// LS Electric XG5000 project: FactoryIO_Automated Warehouse
// PLC LSPLC

PROGRAM NewProgram (task: 스캔 프로그램)

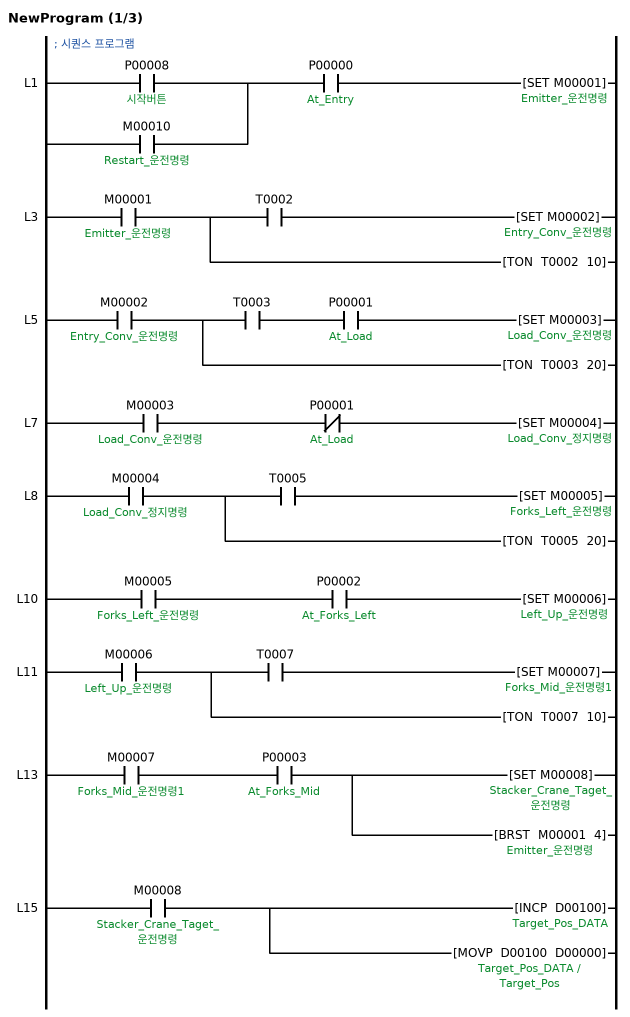
// 시퀀스 프로그램
; L1
LOAD      P00008	// 시작버튼
OR        M00010	// Restart_운전명령
AND       P00000	// At_Entry
SET       M00001	// Emitter_운전명령
; L3
LOAD      M00001	// Emitter_운전명령
MPUSH
AND       T0002
SET       M00002	// Entry_Conv_운전명령
MPOP
TON       T0002 10
; L5
LOAD      M00002	// Entry_Conv_운전명령
MPUSH
AND       T0003
AND       P00001	// At_Load
SET       M00003	// Load_Conv_운전명령
MPOP
TON       T0003 20
; L7
LOAD      M00003	// Load_Conv_운전명령
AND NOT   P00001	// At_Load
SET       M00004	// Load_Conv_정지명령
; L8
LOAD      M00004	// Load_Conv_정지명령
MPUSH
AND       T0005
SET       M00005	// Forks_Left_운전명령
MPOP
TON       T0005 20
; L10
LOAD      M00005	// Forks_Left_운전명령
AND       P00002	// At_Forks_Left
SET       M00006	// Left_Up_운전명령
; L11
LOAD      M00006	// Left_Up_운전명령
MPUSH
AND       T0007
SET       M00007	// Forks_Mid_운전명령1
MPOP
TON       T0007 10
; L13
LOAD      M00007	// Forks_Mid_운전명령1
AND       P00003	// At_Forks_Mid
SET       M00008	// Stacker_Crane_Taget_운전명령
BRST      M00001 4	// Emitter_운전명령
; L15
LOAD      M00008	// Stacker_Crane_Taget_운전명령
INCP      D00100	// Target_Pos_DATA
MOVP      D00100 D00000	// Target_Pos_DATA / Target_Pos

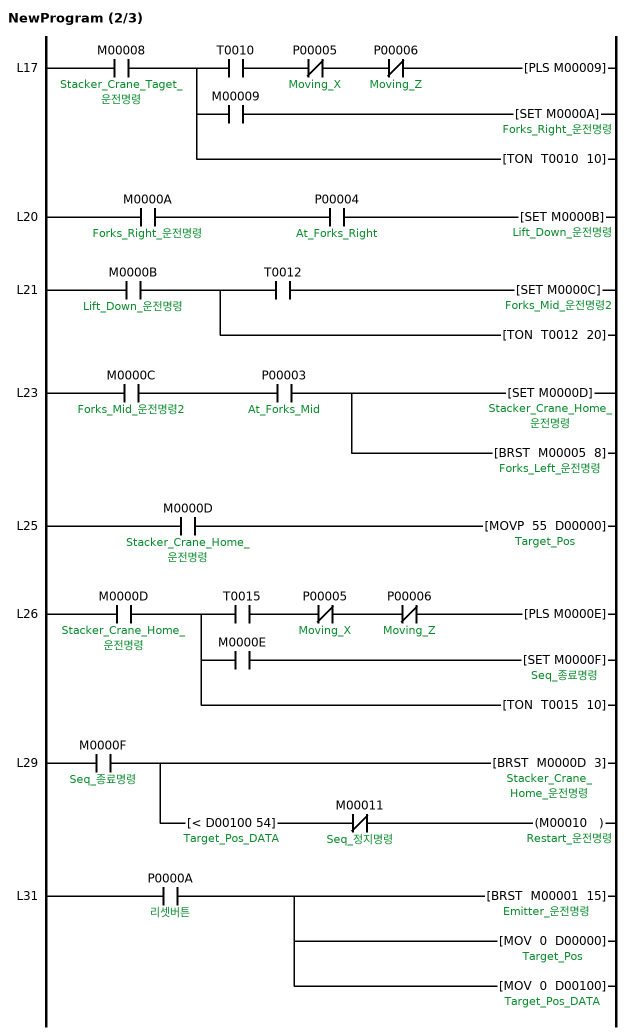
; L17
LOAD      M00008	// Stacker_Crane_Taget_운전명령
MPUSH
AND       T0010
AND NOT   P00005	// Moving_X
AND NOT   P00006	// Moving_Z
OUTP      M00009
MLOAD
AND       M00009
SET       M0000A	// Forks_Right_운전명령
MPOP
TON       T0010 10
; L20
LOAD      M0000A	// Forks_Right_운전명령
AND       P00004	// At_Forks_Right
SET       M0000B	// Lift_Down_운전명령
; L21
LOAD      M0000B	// Lift_Down_운전명령
MPUSH
AND       T0012
SET       M0000C	// Forks_Mid_운전명령2
MPOP
TON       T0012 20
; L23
LOAD      M0000C	// Forks_Mid_운전명령2
AND       P00003	// At_Forks_Mid
SET       M0000D	// Stacker_Crane_Home_운전명령
BRST      M00005 8	// Forks_Left_운전명령
; L25
LOAD      M0000D	// Stacker_Crane_Home_운전명령
MOVP      55 D00000	// Target_Pos
; L26
LOAD      M0000D	// Stacker_Crane_Home_운전명령
MPUSH
AND       T0015
AND NOT   P00005	// Moving_X
AND NOT   P00006	// Moving_Z
OUTP      M0000E
MLOAD
AND       M0000E
SET       M0000F	// Seq_종료명령
MPOP
TON       T0015 10
; L29
LOAD      M0000F	// Seq_종료명령
BRST      M0000D 3	// Stacker_Crane_Home_운전명령
AND<      D00100 54	// Target_Pos_DATA
AND NOT   M00011	// Seq_정지명령
OUT       M00010	// Restart_운전명령
; L31
LOAD      P0000A	// 리셋버튼
BRST      M00001 15	// Emitter_운전명령
MOV       0 D00000	// Target_Pos
MOV       0 D00100	// Target_Pos_DATA

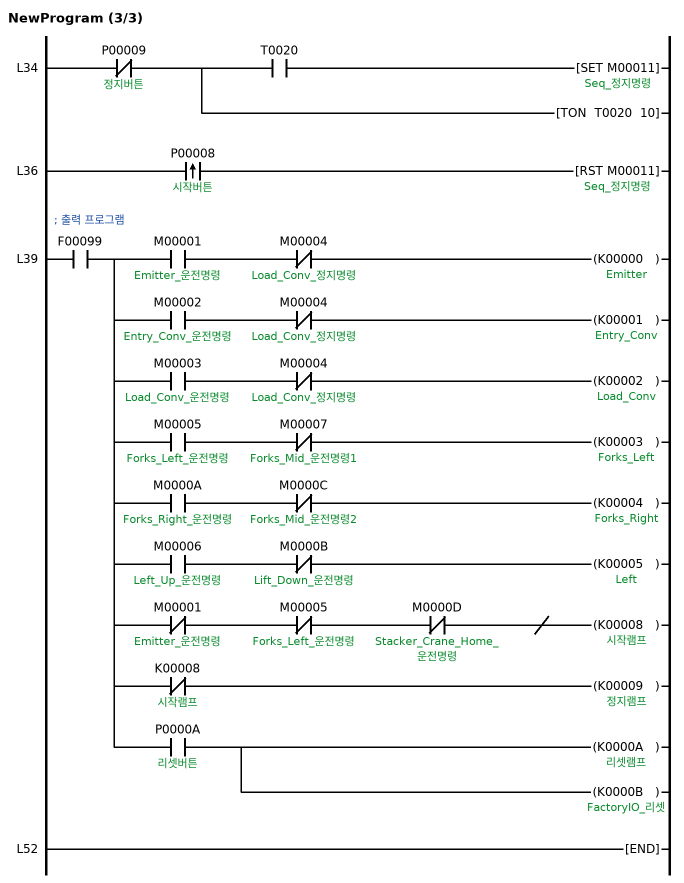
; L34
LOAD NOT  P00009	// 정지버튼
MPUSH
AND       T0020
SET       M00011	// Seq_정지명령
MPOP
TON       T0020 10
; L36
LOADP     P00008	// 시작버튼
RST       M00011	// Seq_정지명령
// 출력 프로그램
; L39
LOAD      F00099
MPUSH
AND       M00001	// Emitter_운전명령
AND NOT   M00004	// Load_Conv_정지명령
OUT       K00000	// Emitter
MLOAD
AND       M00002	// Entry_Conv_운전명령
AND NOT   M00004	// Load_Conv_정지명령
OUT       K00001	// Entry_Conv
MLOAD
AND       M00003	// Load_Conv_운전명령
AND NOT   M00004	// Load_Conv_정지명령
OUT       K00002	// Load_Conv
MLOAD
AND       M00005	// Forks_Left_운전명령
AND NOT   M00007	// Forks_Mid_운전명령1
OUT       K00003	// Forks_Left
MLOAD
AND       M0000A	// Forks_Right_운전명령
AND NOT   M0000C	// Forks_Mid_운전명령2
OUT       K00004	// Forks_Right
MLOAD
AND       M00006	// Left_Up_운전명령
AND NOT   M0000B	// Lift_Down_운전명령
OUT       K00005	// Left
MLOAD
AND NOT   M00001	// Emitter_운전명령
AND NOT   M00005	// Forks_Left_운전명령
AND NOT   M0000D	// Stacker_Crane_Home_운전명령
NOT
OUT       K00008	// 시작램프
MLOAD
AND NOT   K00008	// 시작램프
OUT       K00009	// 정지램프
MPOP
AND       P0000A	// 리셋버튼
OUT       K0000A	// 리셋램프
OUT       K0000B	// FactoryIO_리셋
; L52
END

VARIABLES AND COMMENTS (devices not used above)
M00000	BIT	운전중